FUNCTION_BLOCK FB_AI (* Service Interface Function Block Type *)
  (* Standard: 61499-2 *)
  (* Version 0.0, 2014-5-4, wildai, nxtControl GmbH, template *)
  (* Compiler Cpp nxtControl builtin 1.0 *)
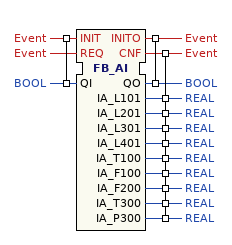
  EVENT_INPUT
    INIT WITH QI; (* Service Initialization *)
    REQ; (* Service Request *)
  END_EVENT
  EVENT_OUTPUT
    INITO WITH QO; (* Initialization Confirm *)
    CNF WITH IA_L101, IA_L201, IA_L301, IA_L401, IA_T100, IA_F100, IA_F200, IA_T300, IA_P300; (* Confirmation of Requested Service *)
  END_EVENT
  VAR_INPUT
    QI : BOOL; (* Event Input Qualifier *)
  END_VAR
  VAR_OUTPUT
    QO : BOOL; (* Event Output Qualifier *)
    IA_L101 : REAL; (* Input data from resource *)
    IA_L201 : REAL;
    IA_L301 : REAL;
    IA_L401 : REAL;
    IA_T100 : REAL;
    IA_F100 : REAL;
    IA_F200 : REAL;
    IA_T300 : REAL;
    IA_P300 : REAL;
  END_VAR
  SERVICE FB_AI/RESOURCE
    SEQUENCE normal_establishment
      FB_AI.INIT+(PARAMS) -> RESOURCE.initialize(PARAMS) -> FB_AI.INITO+();
    END_SEQUENCE
    SEQUENCE unsuccessful_establishment
      FB_AI.INIT+(PARAMS) -> RESOURCE.initialize(PARAMS) -> FB_AI.INITO-(STATUS);
    END_SEQUENCE
    SEQUENCE request_confirm
      FB_AI.REQ+(SD) -> RESOURCE.request(SD) -> FB_AI.CNF+(RD);
    END_SEQUENCE
    SEQUENCE request_inhibited
      FB_AI.REQ-(SD) -> FB_AI.CNF-(STATUS);
    END_SEQUENCE
    SEQUENCE request_error
      FB_AI.REQ+(SD) -> RESOURCE.request(SD) -> FB_AI.CNF-(STATUS);
    END_SEQUENCE
    SEQUENCE indication_response
      FB_AI.RSP(QI,SD) -> RESOURCE.response(QI,SD);
      RESOURCE.indicate(RD) -> FB_AI.IND+(RD);
    END_SEQUENCE
    SEQUENCE indication_inhibited
      RESOURCE.indicate(RD,QI=FALSE) -> RESOURCE.inhibited();
    END_SEQUENCE
    SEQUENCE error_indication
      RESOURCE.error(STATUS) -> FB_AI.IND-(STATUS);
    END_SEQUENCE
    SEQUENCE application_initiated_termination
      FB_AI.INIT-() -> RESOURCE.terminate() -> FB_AI.INITO-(STATUS);
    END_SEQUENCE
    SEQUENCE resource_initiated_termination
      -> FB_AI.INITO-(STATUS);
    END_SEQUENCE
  END_SERVICE
END_FUNCTION_BLOCK
